{attribute 'TcGenerated'}
{attribute 'no-analysis'}
{attribute 'linkalways'}
// This function has been automatically generated from the project information.
VAR_GLOBAL CONSTANT
    {attribute 'const_non_replaced'}
    stLibVersion_KFE_GATT : ST_LibVersion := (iMajor := 0, iMinor := 3, iBuild := 1, iRevision := 0, nFlags := 1, sVersion := '0.3.1');
END_VAR

(* stored: Version 1.1.0.1, ProductVersion 3.1.4022.18
   GVL Global_Version: Id {056414b3-f21d-4496-9751-0a977b7a5984} *)
